PROGRAM G7_Master_Palpages
VAR_INPUT	SFCInit:BOOL;	END_VAR
VAR
	RE_Top_Palp				:R_TRIG;
END_VAR

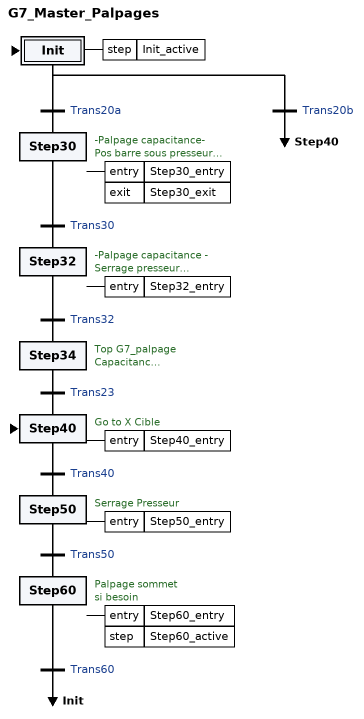
INITIAL_STEP Init:
    Init_active(N);  // step action
END_STEP
TRANSITION FROM Init TO Step30
    := Trans20a;
END_TRANSITION
// -Palpage capacitance-
// Pos barre sous presseurs
// Pour calib capa
// +Go Face 1 réf
STEP Step30:
    Step30_entry(P1);  // entry action
    Step30_exit(P0);  // exit action
END_STEP
TRANSITION FROM Step30 TO Step32
    := Trans30;
END_TRANSITION
// -Palpage capacitance -
// Serrage presseurs
// + XY laser
STEP Step32:
    Step32_entry(P1);  // entry action
END_STEP
TRANSITION FROM Step32 TO Step34
    := Trans32;
END_TRANSITION
// Top G7_palpage
// Capacitance
// (voir Init)
STEP Step34:
END_STEP
TRANSITION FROM Step34 TO Step40
    := Trans23;
END_TRANSITION
TRANSITION FROM Init TO Step40
    := Trans20b;
END_TRANSITION
// Go to X Cible
STEP Step40:
    Step40_entry(P1);  // entry action
END_STEP
TRANSITION FROM Step40 TO Step50
    := Trans40;
END_TRANSITION
// Serrage Presseur
STEP Step50:
    Step50_entry(P1);  // entry action
END_STEP
TRANSITION FROM Step50 TO Step60
    := Trans50;
END_TRANSITION
// Palpage sommet
// si besoin
STEP Step60:
    Step60_entry(P1);  // entry action
    Step60_active(N);  // step action
END_STEP
TRANSITION FROM Step60 TO Init
    := Trans60;
END_TRANSITION

ACTION Init_active:
RE_Top_Palp(clk:=G7_General.Top_Cycles_Palp_Laser);
END_ACTION

ACTION Step30_entry:
 Pos_cible_X := Presseur_Aval_L12.Position_X + Distance_Annulation_Presseur_Laser - Longueur_Barre_en_Pince;	//Après le presseur en aval, 
 Vitesse_Chariot:=Vitesse_Chariot_Auto;
 En_pos_X := FALSE;
 Top_X:=TRUE;
 
 Face_Cible := 1;
 Top_Face:=true;
END_ACTION

ACTION Step30_exit:
Top_face:=false;
END_ACTION

ACTION Step32_entry:
//Serrage presseurs
 Presseur_Amont_K11.Dem_Desserrage:=
 Presseur_Aval_L12.Dem_Desserrage:=FALSE;
 Presseur_Amont_K11.Dem_Serrage:=
 Presseur_Aval_L12.Dem_Serrage:=TRUE;

//Position X et Y Laser
Pos_Cible_X_laser := 190; //Milieu de la course X ?
En_pos_X_Laser:=FALSE;
Top_X_laser:=TRUE;

Pos_Cible_Y_laser := hauteur_aile /2; //Milieu de la cornière
En_pos_Y_Laser:=FALSE;
Top_Y_laser:=TRUE;
END_ACTION

ACTION Step40_entry:
IF  G7_General.Memo_X_Precedent <> Sequence[Pt_Sequence].X THEN
 Pos_Cible_X := Sequence[Pt_Sequence].X;
 En_pos_X:=FALSE;
 Top_x:=TRUE;
END_IF
END_ACTION

ACTION Step5_entry:
Pt_sequence:=Pt_sequence+1;
END_ACTION

ACTION Step50_entry:
IF NOT (Palpage_OK_Face_1 AND Palpage_OK_Face_2) THEN
	Presseur_Amont_K11.Dem_Desserrage:=
	Presseur_Aval_L12.Dem_Desserrage:=FALSE;
	
	Presseur_Amont_K11.Dem_Serrage:=
	Presseur_Aval_L12.Dem_Serrage:=TRUE;
END_IF
END_ACTION

ACTION Step60_active:
IF Palpage_OK_Face_1 AND Palpage_OK_Face_2 THEN
	Top_Palpage_Sommet:=FALSE;
END_IF
END_ACTION

ACTION Step60_entry:
Top_Palpage_Sommet:=true;
END_ACTION

TRANSITION Trans20a:
RE_Top_Palp.Q
AND (Nv_ProcessID 
OR not Prog_Capacitance_Calibration_OK)
END_TRANSITION

TRANSITION Trans20b:
RE_Top_Palp.Q
AND NOT (Nv_ProcessID 
OR NOT Prog_Capacitance_Calibration_OK)
END_TRANSITION

TRANSITION Trans23:
Prog_Capacitance_Calibration_OK
AND NOT Nv_ProcessID
END_TRANSITION

TRANSITION Trans30:
Step30.t > T#20MS
AND En_Pos_X 
AND NOT Top_X

AND Face_En_Pos
AND G7_Sel_Face.init.x
END_TRANSITION

TRANSITION Trans32:
Presseur_Amont_K11.Presseur_EnPlace 
AND Presseur_Aval_L12.Presseur_EnPlace
AND En_pos_X_Laser
AND En_pos_Y_Laser
END_TRANSITION

TRANSITION Trans40:
Step40.t>T#20MS
AND (En_Pos_X
AND NOT Top_X)
OR (Palpage_OK_Face_1 AND Palpage_OK_Face_2)
END_TRANSITION

TRANSITION Trans50:
(Presseur_Amont_K11.Presseur_EnPlace AND Presseur_Aval_L12.Presseur_EnPlace)
OR (Palpage_OK_Face_1 AND Palpage_OK_Face_2)
END_TRANSITION

TRANSITION Trans60:
Step60.t>T#20MS
AND NOT Top_Palpage_Sommet
AND Palpage_OK_Face_1 AND Palpage_OK_Face_2
AND Prog_Capacitance_Calibration_OK AND NOT Nv_ProcessID
END_TRANSITION

END_PROGRAM

(* stored: Version 1.1.0.1, ProductVersion 3.1.4024.15
   POU G7_Master_Palpages: Id {7f42b02b-01ca-43ab-93fb-ff09daaa10ea}, SpecialFunc None
   Action Init_active: Id {9940c74c-16fb-4dca-96f2-b20baaa27420}
   Action Step30_entry: Id {05b496a1-9845-41ce-8801-5c198b199d52}
   Action Step30_exit: Id {f0be1e73-6658-4364-818e-905386529db2}
   Action Step32_entry: Id {4e13aff4-2e0f-4b89-8782-f97c6f4c4e1e}
   Action Step40_entry: Id {f0538d28-f1a7-4c33-9400-718c62f895c2}
   Action Step5_entry: Id {410ae23a-c28e-4ec8-94b0-8eb024cc41c6}
   Action Step50_entry: Id {9ba0f542-ddac-4afb-9d52-85f02e7244f8}
   Action Step60_active: Id {9b36859f-af3a-4d04-ba9b-ba56d80a9ac1}
   Action Step60_entry: Id {afb8e265-b6eb-41a4-9c99-2e759c226308}
   Transition Trans20a: Id {01fa4212-2f4b-40ba-878d-8f4dcbb8d001}
   Transition Trans20b: Id {1540734c-8c13-4ef4-bd4a-da421aef29e4}
   Transition Trans23: Id {3ad6e847-c947-4f64-9ec2-c43f305c8259}
   Transition Trans30: Id {99b8f2e9-e720-4916-a7c2-7d834371177b}
   Transition Trans32: Id {f562fe78-314e-4f0b-932b-3f30c2241ea7}
   Transition Trans40: Id {04db96fa-c186-4289-82e0-b48a6d6e8b81}
   Transition Trans50: Id {795923d3-7278-4e3c-8c68-12c76f2242e1}
   Transition Trans60: Id {07618f17-f8aa-4bd6-96bc-289c37338962} *)
